FUNCTION CONCAT3 : STRING
VAR_INPUT
	STR1	: STRING;
	STR2	: STRING;
	STR3	: STRING;
END_VAR
VAR
	sTemp	: STRING;
END_VAR

sTemp := CONCAT(STR1,STR2);
sTemp := CONCAT(sTemp, STR3);
CONCAT3 := sTemp;

END_FUNCTION

(* stored: Version 1.1.0.1, ProductVersion 3.1.4024.12
   POU CONCAT3: Id {e91f96f3-110c-44cb-add4-a051574eb139}, SpecialFunc None *)
